TYPE P2_AxiseNo ://伺服轴号、虚轴号
STRUCT
	AxisName:ST_AxisName;//伺服轴号
	VirAxisName:ST_VirAxisName;//虚轴号
END_STRUCT
END_TYPE

(* stored: Version 1.1.0.1, ProductVersion 3.1.4024.9
   DUT P2_AxiseNo: Id {b53fb129-6338-41ce-b7af-11cd0629994b} *)
